{attribute 'GeneratedUsingTerminal: KL9505-0010'}
{attribute addProperty BoxType "KL9505-0010"}
{attribute addProperty Id "Diag_1AT %I*Diag_1F4F45730"}
{attribute addProperty CRC "3837602616"}
{attribute addProperty Size "0"}
TYPE KL_E4BD2B38 :
STRUCT
	{attribute addProperty Name "Diag_1"}
	Diag_1 : Diag_1F4F4573;
END_STRUCT
END_TYPE

(* stored: Version 1.2.0.0, ProductVersion 3.1.4024.9
   DUT KL_E4BD2B38: Id {80f2913a-dc0e-4b3c-936f-acb8e3160892} *)
